{attribute 'GeneratedUsingTerminal: EL2595-0000-0018'}
{attribute addProperty BoxType "EL2595-0000-0018"}
{attribute addProperty Id "ControlAT %Q*Control_7648F4323"}
{attribute addProperty CRC "1976945122"}
{attribute addProperty Size "3"}
TYPE DOX_Control_75D5C9E2 EXTENDS OutputBase_10CEE7DE :
STRUCT
	{attribute addProperty Name "Control"}
	Control AT %Q* : Control_7648F432;
END_STRUCT
END_TYPE

(* stored: Version 1.2.0.0, ProductVersion 3.1.4024.9
   DUT DOX_Control_75D5C9E2: Id {7806d641-b384-4391-a0bd-8b5190a0faa8} *)
